{attribute 'qualified_only'}
VAR_GLOBAL
	// status variables
	opened		: BOOL;
	closed		: BOOL;
	opening		: BOOL;
	closing		: BOOL;
	stopped		: BOOL;
	error		: BOOL;
	
	// commands
	open		: BOOL;
	close		: BOOL;
	stop		: BOOL;
	reset		: BOOL;
END_VAR

(* stored: Version 1.1.0.1, ProductVersion 3.1.4024.12
   GVL GVL_Roof: Id {36ac59c0-875c-4faa-b3fd-660f48a145a6} *)
